{region '#Template'}
	{attribute 'Version' := '1.0.0.0'}
	{attribute 'Tags' := '"LCID": "1031", "Text": "Universal, Control, Timer"'}
	{attribute 'Tags' := '"LCID": "1033", "Text": "Universal, Control, Timer"'}
	{attribute 'Description' := '"LCID": "1031", "Text": "Zeitglied Einschaltverzögert"'}
	{attribute 'Description' := '"LCID": "1033", "Text": "Timer switch-on delayed"'}
{endregion}
FUNCTION_BLOCK FB_BA_DlyOn EXTENDS FB_BA_View
VAR_INPUT
	bVal					: BOOL;	
END_VAR
VAR_OUTPUT
	bQ						: BOOL;
	nRT						: UDINT;// Restzeit [s] // remaining time [s]	
END_VAR
VAR_INPUT CONSTANT
	TiDly					: FB_BA_AV_Op;		
END_VAR	
VAR	
	tonDlyOn				: TON;
END_VAR
VAR // added by the converter: edge detectors and wires of the graphical bodies
    _w1, _w2 : ANY;
END_VAR

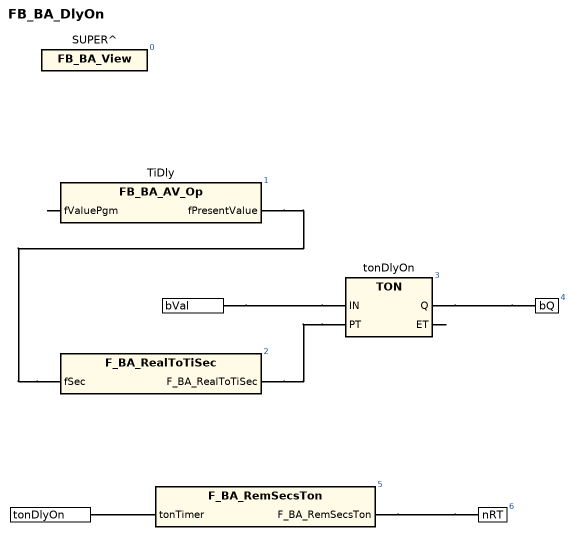
SUPER^(); // FB_BA_View
TiDly(); // FB_BA_AV_Op
_w1 := F_BA_RealToTiSec(fSec := TiDly.fPresentValue);
tonDlyOn(IN := bVal, PT := _w1); // TON
bQ := tonDlyOn.Q;
_w2 := F_BA_RemSecsTon(tonTimer := tonDlyOn);
nRT := _w2;

METHOD FB_init : BOOL
VAR_INPUT
	bInitRetains : BOOL; // if TRUE, the retain variables are initialized (warm start / cold start)
	bInCopyCode : BOOL;  // if TRUE, the instance afterwards gets moved into the copy code (online change)
END_VAR
TiDly.iParent			:= THIS^;
TiDly.iLabel			:= LblUniControl.DelayOn_TiDly;		 
TiDly.sObjectName		:= '{Idx=01}';								 	 
TiDly.eUnit 			:= E_BA_Unit.eTime_Seconds;								 
TiDly.fValueRm			:= 0;		
TiDly.fCOVIncrement		:= BA2_Param.fDefCOVIncrement;
END_METHOD

END_FUNCTION_BLOCK

(* stored: Version 1.1.0.1, ProductVersion 3.1.4024.9
   POU FB_BA_DlyOn: Id {d2230bbe-62fa-48d4-8a3f-5e521edffba1}, SpecialFunc None
   Method FB_init: Id {b566bcb5-2ae1-4fbf-a016-8fec367f260c} *)
